// TIA Portal V17 export
// export: Created 2023-12-22T15:04:41.8216576Z, ExportSetting WithDefaults, DisplayName Totally Integrated Automation Portal, DisplayVersion V17, DisplayName TIA Portal Openness, DisplayVersion V17, DisplayName TIA Portal Version Control Interface, DisplayVersion V17, DisplayName STEP 7 Professional, DisplayVersion V17, DisplayName STEP 7 Safety, DisplayVersion V17, DisplayName WinCC Advanced, DisplayVersion V17
DATA_BLOCK "PE_1_DB"   // DB304
VERSION : 0.1
// stored: AutoNumber false, DBAccessibleFromOPCUA true, InstanceOfName AI_ex, InstanceOfType FB
"AI_ex"
   // VAR_OUTPUT
   //    S_Alarm : Bool;
   // END_VAR
   // VAR_IN_OUT
   //    Signal : Int;
   //    Result : Real;
   // END_VAR
   // VAR RETAIN
   //    CMD : "CMD";
   //    Mode : Int;
   //    Status : Int;
   //    Use : Struct
   //       RTD { S7_SetPoint := 'True'} : Bool := FALSE;
   //       Filter { S7_SetPoint := 'True'} : Bool := FALSE;
   //       Inverse { S7_SetPoint := 'True'} : Bool := FALSE;
   //       Indirect { S7_SetPoint := 'True'} : Bool := TRUE;
   //       Status { S7_SetPoint := 'True'} : Bool := FALSE;
   //       Light { S7_SetPoint := 'True'} : Bool := FALSE;
   //       Lim_Low { S7_SetPoint := 'True'} : Bool := TRUE;
   //       Lim_High { S7_SetPoint := 'True'} : Bool := FALSE;
   //       Communication { S7_SetPoint := 'True'} : Bool := FALSE;
   //    END_STRUCT;
   //    VmA : Real;
   //    RTD_c { S7_SetPoint := 'True'} : Real := 10.0;
   //    Calibration { S7_SetPoint := 'True'} : Real := 0.0;
   //    Converter { S7_SetPoint := 'True'} : "Converter_LAD";
   //    SP : Struct
   //       NC { S7_SetPoint := 'True'} : Real := -500.0;
   //       SC { S7_SetPoint := 'True'} : Real := 32000.0;
   //       HH { S7_SetPoint := 'True'} : Real := 6.0;
   //       H { S7_SetPoint := 'True'} : Real := 5.0;
   //       L { S7_SetPoint := 'True'} : Real := 0.0;
   //       LL { S7_SetPoint := 'True'} : Real := -0.5;
   //    END_STRUCT;
   //    Tx { S7_SetPoint := 'True'} : Array[0..5] of "Time_R";
   //    Alarm : Struct
   //       ST : Bool;
   //       HH : Bool;
   //       H : Bool;
   //       L : Bool;
   //       LL : Bool;
   //       NC : Bool;
   //       SC : Bool;
   //    END_STRUCT;
   //    Alarms : Word;
   //    Events : Word;
   //    pos : Array[0..15] of Bool;
   //    Input_Type { S7_SetPoint := 'True'} : Int := 0;
   //    CodeID { S7_SetPoint := 'True'} : Int := 0;
   //    "Type" { S7_SetPoint := 'True'} : Int := 0;
   //    ADDR { S7_SetPoint := 'True'} : Int := 260;
   //    Filter_SP { S7_SetPoint := 'True'} : Int := 100;
   //    "Name" { S7_SetPoint := 'True'} : String[5] := 'PE 23';
   //    Filter_DB : "Filter";
   //    Time_DTL { S7_SetPoint := 'True'} : DTL := DTL#2012-01-22-23:24:12.764341;
   // END_VAR
BEGIN
   Converter.Use_Min_In := FALSE;
   Converter.Use_Max_In := FALSE;
   Converter.Use_Min_Out := FALSE;
   Converter.Use_Max_Out := FALSE;
   Converter.IO := FALSE;
   Converter.Inverse := FALSE;
   Converter.Min_In := 0.0;
   Converter.Min_Out := 0.0;
   Converter.Max_In := 27648.0;
   Converter.Max_Out := 16.0;
   Tx[0..1].SP := 3.0;
   Tx[2..5].SP := 1.0;
   Tx[0..5].One := 0.1;
END_DATA_BLOCK
